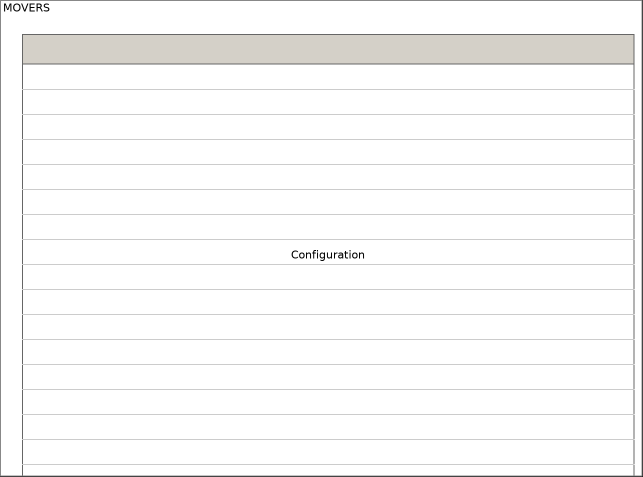
VISUALIZATION VI_XTSMoversVisu  // 643x477
VAR_IN_OUT
	xts : XTS_System;
END_VAR
VAR
	stTableStruct : ARRAY [1..25] OF stTableStructx10;
END_VAR
    Rectangle (0,0 643x477), "MOVERS"
    Table (22,34 612x442), "Configuration", data array: stTableStruct
        p3854506369: xts.ax[INDEX].ax.NcToPlc.AxisId
        p1892666644: xts.ax[INDEX].ax.NcToPlc.ModuloSetPos
        p338671338: xts.ax[INDEX].ax.NcToPlc.SetVelo
        p2170511999: xts.ax[INDEX].ax.Status.MotionState
        p3723444502: xts.ax[INDEX].ax.NcToPlc.ErrorCode
        p2232123230: Name
        p511219082: Position
        p1755163831: Velocity
        p2237128397: Error ID
        p505689113: Process Time
        p1757482276: Stop Positions
        p4088588272: Ack Mode
        p2243050616: Disable
        p516019884: Travel Time
        p2685023577: stTableStruct.b1
        p3312258591: stTableStruct.b2
        p1791247317: stTableStruct.b3
        p262371475: stTableStruct.b4
        p4008173056: stTableStruct.b5
        p2340480326: stTableStruct.b6
        p606709900: stTableStruct.b7
        p1095668682: stTableStruct.b8
        p1037165547: stTableStruct.b9
        p1488378029: stTableStruct.b10
        Columns.Column.[3].Template: OnMouseClick: write the text variable via Default
        Columns.Column.[8].Template: xts.aStations[INDEX].stCfg.bDisable=true; toggle xts.aStations[INDEX].stCfg.bDisable
        Columns.Column.[6].Template: OnMouseClick: write the text variable via Default, min 1, max 3
        Columns.Column.[4].Template: OnMouseClick: write the text variable via Default
        Columns.Column.[5].Template: OnMouseClick: write the text variable via Default
        Columns.Column.[0].Template: OnMouseClick: OpenDialog Dialog=Mover_VISU, Parameters={fbMover: xts.aMovers[INDEX]}, OpenModal=True, OpenCentered=True
        Columns.Column.[7].Template: OnMouseClick: write the text variable via Default
        Columns.Column.[9].Template: OnMouseClick: write the text variable via Default
END_VISUALIZATION

(* stored: Version 1.1.0.1, ProductVersion 3.1.4024.11
   Visu VI_XTSMoversVisu: Id {91fbc901-a7c8-4f77-a3e0-550592c41db5} *)
